(* PLC project servo_mode, Dassault Systèmes ControlBuild 2024x *)
(* stored: creationDateTime 2023-10-04T11:03:55-01:00 *)

(* This module managed the priority between local and remote commands *)
FUNCTION_BLOCK motion_control.servo_mode
  VAR_INPUT
    PLC_StatusReady : BOOL := true;
    PLC_StatusMoved : BOOL := false;
    PLC_StatusStand : BOOL := false;
    PLC_ActualPositionAx : REAL := 0.0;
    PLC_ActualPositionMa : REAL := 0.0;
    PLC_ActualVelocity : REAL := 0.0;
  END_VAR
  VAR_INPUT
    StatusReady : BOOL := true;
    StatusMoved : BOOL := false;
    StatusStand : BOOL := false;
    ActualPositionMa : REAL := 0.0;
    ActualVelocity : REAL := 0.0;
    MaximumVelocity : REAL := 0.0;
  END_VAR
  VAR_INPUT
    physicalPosInit : REAL := 0.0;
  END_VAR
  VAR_IN_OUT
    ActualPositionAx : REAL := 0.0;
  END_VAR
  VAR_OUTPUT
    StatusReady_o : BOOL := true;
    StatusMoved_o : BOOL := false;
    StatusStand_o : BOOL := false;
    ActualPositionAx_o : REAL := 0.0;
    ActualPositionMa_o : REAL := 0.0;
    ActualVelocity_o : REAL := 0.0;
    MaximumVelocity_o : REAL := 0.0;
    StatusPosIncrease_o : BOOL := false;
    StatusPosDecrease_o : BOOL := false;
    displayJauge_o : REAL := 0.0;
  END_VAR
  VAR
    PLCMode : BOOL := false;
    PLCMode1 : BOOL := false;
    initDone : BOOL := false;
    displayPosMin : REAL := 0.0;
    displayPosMax : REAL := 0.0;
    PLC_ActualPositionAx1 : REAL := 0.0;
    PLC_ActualVelocity1 : REAL := 0.0;
    ActualPositionAx1 : REAL := 0.0;
    ActualVelocity1 : REAL := 0.0;
    offsetAxToMa : REAL := 0.0;
    offsetAxToMa1 : REAL := 0.0;
    ActualPositionMa_o1 : REAL := 0.0;
  END_VAR


ACTION C_source_code:
if (!initDone) {
	PLC_ActualPositionAx = physicalPosInit;
	PLC_ActualPositionMa = physicalPosInit;
	ActualPositionAx = physicalPosInit;
	ActualPositionMa = physicalPosInit;
} else {
	if (PLC_ActualPositionAx1 != PLC_ActualPositionAx) PLCMode = 1;
	if (PLC_ActualVelocity1 != PLC_ActualVelocity) PLCMode = 1;
	if (ActualPositionAx1 != ActualPositionAx) PLCMode = 0;
	if (ActualVelocity1 != ActualVelocity) PLCMode = 0;
	if (PLCMode != PLCMode1) {
		if (PLCMode == 0) ActualPositionAx = PLC_ActualPositionAx;
	}
	PLCMode1 = PLCMode;
}

// modification of ref position
if (offsetAxToMa != offsetAxToMa1) {
	displayPosMax += (offsetAxToMa - offsetAxToMa1);
	displayPosMin += (offsetAxToMa - offsetAxToMa1);
}

if (PLCMode) {
	StatusReady_o = PLC_StatusReady;
	StatusMoved_o = (PLC_StatusStand == 0);
	StatusStand_o = PLC_StatusStand;
	ActualPositionAx_o = PLC_ActualPositionAx;
	ActualPositionMa_o = PLC_ActualPositionMa;
	ActualVelocity_o = PLC_ActualVelocity;
	MaximumVelocity_o = MaximumVelocity;
} else {
	StatusReady_o = StatusReady;
	StatusMoved_o = StatusMoved;
	StatusStand_o = StatusStand;
	ActualPositionAx_o = ActualPositionAx;
	ActualPositionMa_o = ActualPositionMa;
	ActualVelocity_o = ActualVelocity;
	MaximumVelocity_o = MaximumVelocity;
}


// DISPLAY CALC
if (initDone == 0) {
	displayPosMax = ActualPositionMa_o;
	displayPosMin = ActualPositionMa_o;
}
if (ActualPositionMa_o1 != ActualPositionMa_o) {
	if (ActualPositionMa_o > displayPosMax) {
		displayPosMax = ActualPositionMa_o;
		displayJauge_o = 100*(ActualPositionMa_o - displayPosMin)/(displayPosMax - displayPosMin);
	} else {
		if (ActualPositionMa_o < displayPosMin) {
			displayPosMin = ActualPositionMa_o;
			displayJauge_o = 100 - 100*(displayPosMax - ActualPositionMa_o )/(displayPosMax - displayPosMin);
		} else {
			if (displayPosMax != displayPosMin) displayJauge_o = 100*(ActualPositionMa_o - displayPosMin)/(displayPosMax - displayPosMin);
		}
	}
}


if (ActualVelocity_o > 0.0) StatusPosIncrease_o = 1; else StatusPosIncrease_o = 0;
if (ActualVelocity_o < 0.0) StatusPosDecrease_o = 1; else StatusPosDecrease_o = 0;

offsetAxToMa1 = offsetAxToMa;

PLC_ActualPositionAx1 = PLC_ActualPositionAx;
PLC_ActualVelocity1 = PLC_ActualVelocity;
ActualPositionAx1 = ActualPositionAx;
ActualVelocity1 = ActualVelocity;

initDone = 1;
END_ACTION
END_FUNCTION_BLOCK
